// SIMATIC STEP 7 (V5.x) project Ножницы №2(гитльотина)
// CPU: CPU 312C
// station: Hardware
// station: SIMATIC 300(1)
// station: P_ADR_BUS
// program: S7 Program(2)

SYMBOL_TABLE
"Автоматический режим"	FC 1	FC 1
"Режим наладки"	FC 2	FC 2
"S1.1"	I 0.0	BOOL	// Нижнее положение стола
"S1.2-S1.5"	I 0.1	BOOL	// Верхнее положение стола
"S1.6"	I 0.2	BOOL	// подача стола вверх
"S3.1-S3.3"	I 0.3	BOOL	// Кнопки СТОП
"S3.4"	I 0.4	BOOL	// ПУСК стол вверх
"S3.5"	I 0.5	BOOL	// ПУСК стол вниз
"S3.6"	I 0.6	BOOL	// СТОП вакуум на подающем столе
"S3.8"	I 0.7	BOOL	// ПУСК вакуум на подающем столе
"S3.10-S3.10a"	I 1.0	BOOL	// ПУСК привод
"S3.11-S3.11a"	I 1.1	BOOL	// СТОП привод
"S3.12-S3.12a"	I 1.2	BOOL	// ВКЛ.муфта на гильотине
"S3.13-S3.14a"	I 1.3	BOOL	// ОТКЛ. муфта
"B8.1"	I 1.4	BOOL	// Стол(наличие металла)
"B8.2"	I 1.5	BOOL	// Вакуум   (фаза)
"B8.3"	I 1.6	BOOL	// Двойной лист
"S1.7-S1.9"	I 1.7	BOOL	// Блокировка гильотины.
"S3.7-S3.7a"	I 124.0	BOOL	// СТОП Вакуум на гильотине
"S3.9"	I 124.1	BOOL	// ПУСК Вакуум на гильотине слева
"S3.9a"	I 124.2	BOOL	// ПУСК Вакуум на гильотине справа
"S4.1"	I 124.3	BOOL	// Переключатель РУЧН.-АВТ.
"S3.15-S3.16"	I 124.4	BOOL	// ВКЛ Муфта на середине стола
"m0.0"	M 0.0	BOOL	// Нижнее положение стола.
"m0.1"	M 0.1	BOOL	// Верхнее положение стола.
"m0.2"	M 0.2	BOOL	// Меркер наличия металла.
"Организационный блок"	OB 1	OB 1
"K9.1"	Q 4.0	BOOL	// Стол вниз
"K9.1а"	Q 4.1	BOOL	// Стол вверх
"K9.2"	Q 4.2	BOOL	// Вакуум
"K9.3"	Q 4.3	BOOL	// Привод
"Y1.2"	Q 4.4	BOOL	// Выбрасыватель двойных листов
"Y1.3"	Q 4.5	BOOL	// Воздух раздувки листов
"K9.4"	Q 4.6	BOOL	// Муфта
END_SYMBOL_TABLE

FUNCTION "Автоматический режим" : VOID	// FC 1
VERSION : 0.1
BEGIN
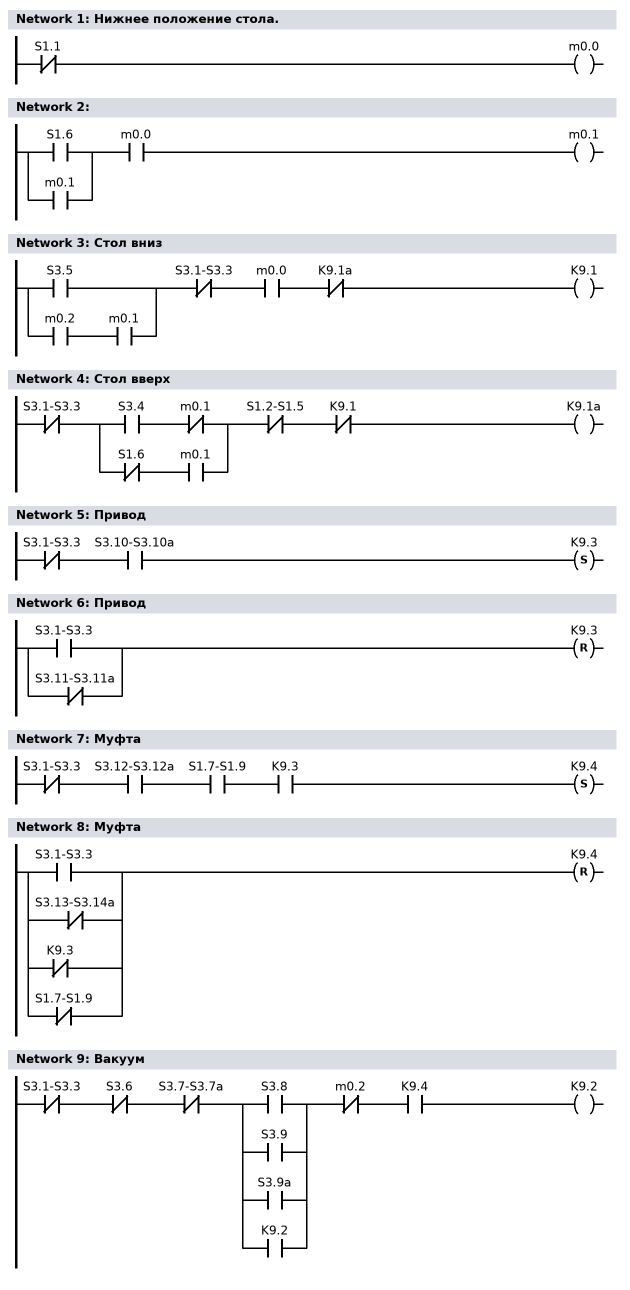
NETWORK
TITLE = Нижнее положение стола.
//Меркер нижнего положения стола.
      AN    "S1.1";
      =     "m0.0";
NETWORK
TITLE =
      A(;
      O     "S1.6";
      O     "m0.1";
      );
      A     "m0.0";
      =     "m0.1";
NETWORK
TITLE = Стол вниз
      A(;
      O     "S3.5";
      O;
      A     "m0.2";
      A     "m0.1";
      );
      AN    "S3.1-S3.3";
      A     "m0.0";
      AN    "K9.1а";
      =     "K9.1";
NETWORK
TITLE = Стол вверх
      AN    "S3.1-S3.3";
      A(;
      A     "S3.4";
      AN    "m0.1";
      O;
      AN    "S1.6";
      A     "m0.1";
      );
      AN    "S1.2-S1.5";
      AN    "K9.1";
      =     "K9.1а";
NETWORK
TITLE = Привод
      AN    "S3.1-S3.3";
      A     "S3.10-S3.10a";
      S     "K9.3";
NETWORK
TITLE = Привод
      O     "S3.1-S3.3";
      ON    "S3.11-S3.11a";
      R     "K9.3";
NETWORK
TITLE = Муфта
      AN    "S3.1-S3.3";
      A     "S3.12-S3.12a";
      A     "S1.7-S1.9";
      A     "K9.3";
      S     "K9.4";
NETWORK
TITLE = Муфта
      O     "S3.1-S3.3";
      ON    "S3.13-S3.14a";
      ON    "K9.3";
      ON    "S1.7-S1.9";
      R     "K9.4";
NETWORK
TITLE = Вакуум
      AN    "S3.1-S3.3";
      AN    "S3.6";
      AN    "S3.7-S3.7a";
      A(;
      O     "S3.8";
      O     "S3.9";
      O     "S3.9a";
      O     "K9.2";
      );
      AN    "m0.2";
      A     "K9.4";
      =     "K9.2";
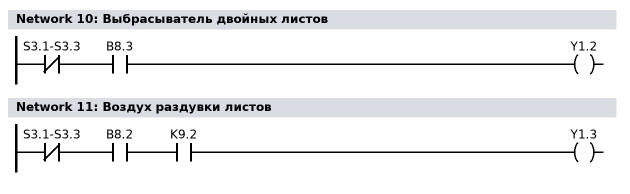
NETWORK
TITLE = Выбрасыватель двойных листов
      AN    "S3.1-S3.3";
      A     "B8.3";
      =     "Y1.2";
NETWORK
TITLE = Воздух раздувки листов
      AN    "S3.1-S3.3";
      A     "B8.2";
      A     "K9.2";
      =     "Y1.3";
END_FUNCTION

FUNCTION "Режим наладки" : VOID	// FC 2
VERSION : 0.1
BEGIN
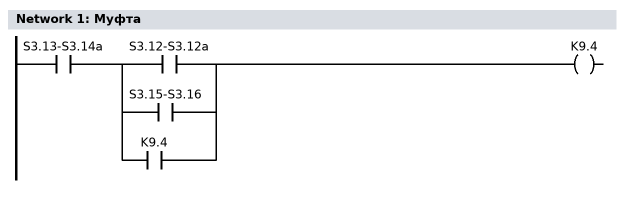
NETWORK
TITLE = Муфта
      A     "S3.13-S3.14a";
      A(;
      O     "S3.12-S3.12a";
      O     "S3.15-S3.16";
      O     "K9.4";
      );
      =     "K9.4";
END_FUNCTION

ORGANIZATION_BLOCK "Организационный блок"	// OB 1
TITLE = "Main Program Sweep (Cycle)"
VERSION : 0.1
VAR_TEMP
  OB1_EV_CLASS : BYTE ;	//Bits 0-3 = 1 (Coming event), Bits 4-7 = 1 (Event class 1)
  OB1_SCAN_1 : BYTE ;	//1 (Cold restart scan 1 of OB 1), 3 (Scan 2-n of OB 1)
  OB1_PRIORITY : BYTE ;	//Priority of OB Execution
  OB1_OB_NUMBR : BYTE ;	//1 (Organization block 1, OB1)
  OB1_RESERVED_1 : BYTE ;	//Reserved for system
  OB1_RESERVED_2 : BYTE ;	//Reserved for system
  OB1_PREV_CYCLE : INT ;	//Cycle time of previous OB1 scan (milliseconds)
  OB1_MIN_CYCLE : INT ;	//Minimum cycle time of OB1 (milliseconds)
  OB1_MAX_CYCLE : INT ;	//Maximum cycle time of OB1 (milliseconds)
  OB1_DATE_TIME : DATE_AND_TIME ;	//Date and time OB1 started
END_VAR
BEGIN
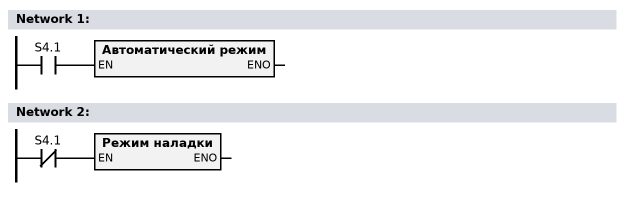
NETWORK
TITLE =
      A     "S4.1";
      JNB   _001;
      CALL  "Автоматический режим";
_001: NOP   0;
NETWORK
TITLE =
      AN    "S4.1";
      JNB   _002;
      CALL  "Режим наладки";
_002: NOP   0;
END_ORGANIZATION_BLOCK
